(* CODESYS project setReset.project

Project tree, tasks and I/O mapping:
  Device : CODESYS Control Win V3, 3S - Smart Software Solutions GmbH, order no. 305021, version 3.5.8.10
    application Application
      libraries: Standard, * (System)
      task MainTask (cyclic, interval t#20ms, priority 1) calls PLC_PRG
      task VISU_TASK (cyclic, interval 100 ms, priority 31) calls VisuElems.Visu_Prg
      program PLC_PRG [LD]
      visualisation Visualization
  libraries: VisuSymbols, 3.5.8.0 (System)
  text list GlobalTextList
*)

// Device/Application/PLC_PRG
PROGRAM PLC_PRG
VAR
	set: BOOL;
	czerwona: BOOL;
	zielona: BOOL;
	niebieska: BOOL;
	zolta: BOOL;
	reset: BOOL;
END_VAR

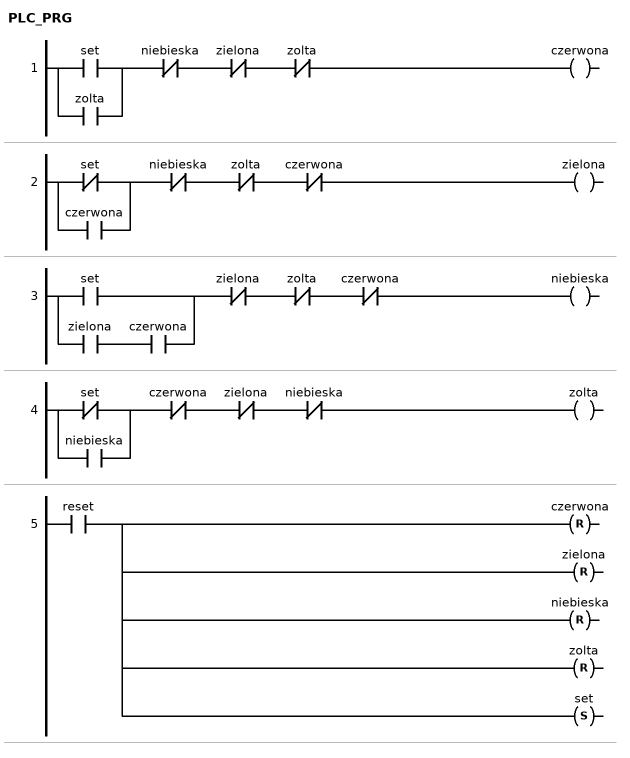
// NETWORK 1
czerwona := (set OR zolta) AND NOT niebieska AND NOT zielona AND NOT zolta;

// NETWORK 2
zielona := (NOT set OR czerwona) AND NOT niebieska AND NOT zolta AND NOT czerwona;

// NETWORK 3
niebieska := (set OR zielona AND czerwona) AND NOT zielona AND NOT zolta AND NOT czerwona;

// NETWORK 4
zolta := (NOT set OR niebieska) AND NOT czerwona AND NOT zielona AND NOT niebieska;

// NETWORK 5
czerwona R= reset;
zielona R= reset;
niebieska R= reset;
zolta R= reset;
set S= reset;

END_PROGRAM

// Device/Application/Visualization
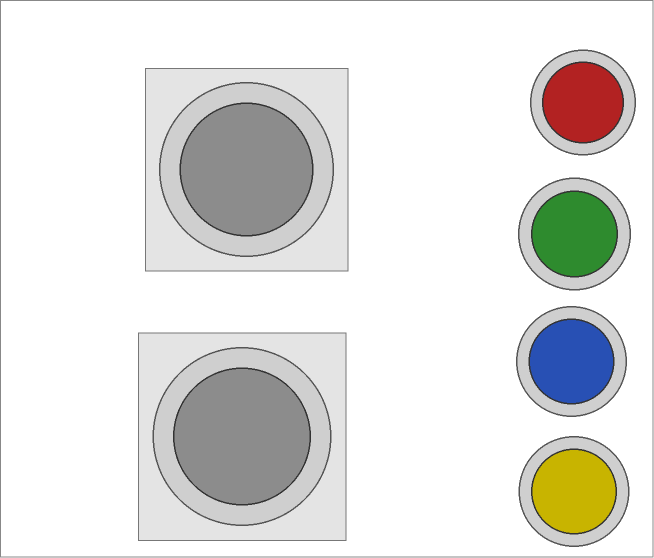
VISUALIZATION Visualization  // 654x558
    PushSwitch (139,68 215x203), variable: PLC_PRG.set, behaviour: TOGGLE, style: Switch-PushSwitch-Gray
    PushSwitch (138,329 208x215), variable: PLC_PRG.reset, behaviour: TOGGLE, style: Switch-PushSwitch-Gray
    Lamp1 (505,297 133x129), variable: PLC_PRG.niebieska, style: Lamp-Lamp1-Blue
    Lamp1 (507,427 134x129), variable: PLC_PRG.zolta, style: Lamp-Lamp1-Yellow
    Lamp1 (509,165 131x138), variable: PLC_PRG.zielona, style: Lamp-Lamp1-Green
    Lamp1 (514,41 138x123), variable: PLC_PRG.czerwona, style: Lamp-Lamp1-Red
END_VISUALIZATION
